(* CODESYS project GVL_MAGAZINE.gvl.xml

Project tree, tasks and I/O mapping:
  global variables GVL_MAGAZINE
*)

// GVL_MAGAZINE
{attribute 'qualified_only'}
VAR_GLOBAL
	AutoCommand : ST_MAGAZINE_COMMAND; // Автоматическая команда магазину
	Command : ST_ROBOT_COMMAND; // Команда роботу от магазина
	Status  : ST_MAGAZINE_STATUS; // Рабочие статусы магазина
	Diag    : ST_MAGAZINE_DIAG; // Состояние автомата магазина
	Error   : ST_MAGAZINE_ERRORS; // Ошибки магазина
END_VAR
